(* Logix 5000 project; controller ABB_Drive_Test vendor 1 type 14 code 149 rev 33.12; software revision 33.01; part 6 of 6 *)
(* tags used below, declared in another part *)
   flagDesAcell : BOOL;   // Flag Auxiliar Boton de Parada
   indiceLocal : DINT;
   InicioDinagram : BOOL;   // Inicio de la Adquisión del Dinagrama
   numeroMuestras : DINT;   // Numero de Muestras del Stroke
   pausa : BOOL;
   rpmFeedback : INT;   // Valor absoluto de la referencia 0 no lo toma
   VCarga : REAL[1500];
   Vct : REAL[1500];
   VPosicion : REAL[1500];   // vector de potencia por comunicación
   VPotencia : REAL[1500];
   VPotenciaC : REAL[1500];   // Vector de potencia cableado
   VProximetro : BOOL[1504];
   ABB_GetAtt_Value : DINT;
   ABB_GetMsg : MESSAGE;
   ABB_Input : ABB_Read;
   ABB_Msg_SetValue : DINT;
   ABB_Output : ABB_Write;
   ABB_SetMsg : MESSAGE;
   counters : COUNTER[20];
   Proximetro : BOOL;
   SWC : SWC;
   Timmers : TIMER[10];
(* T000_MainProgram, continued *)

ROUTINE R001_ABB_Drive   (* ladder *)
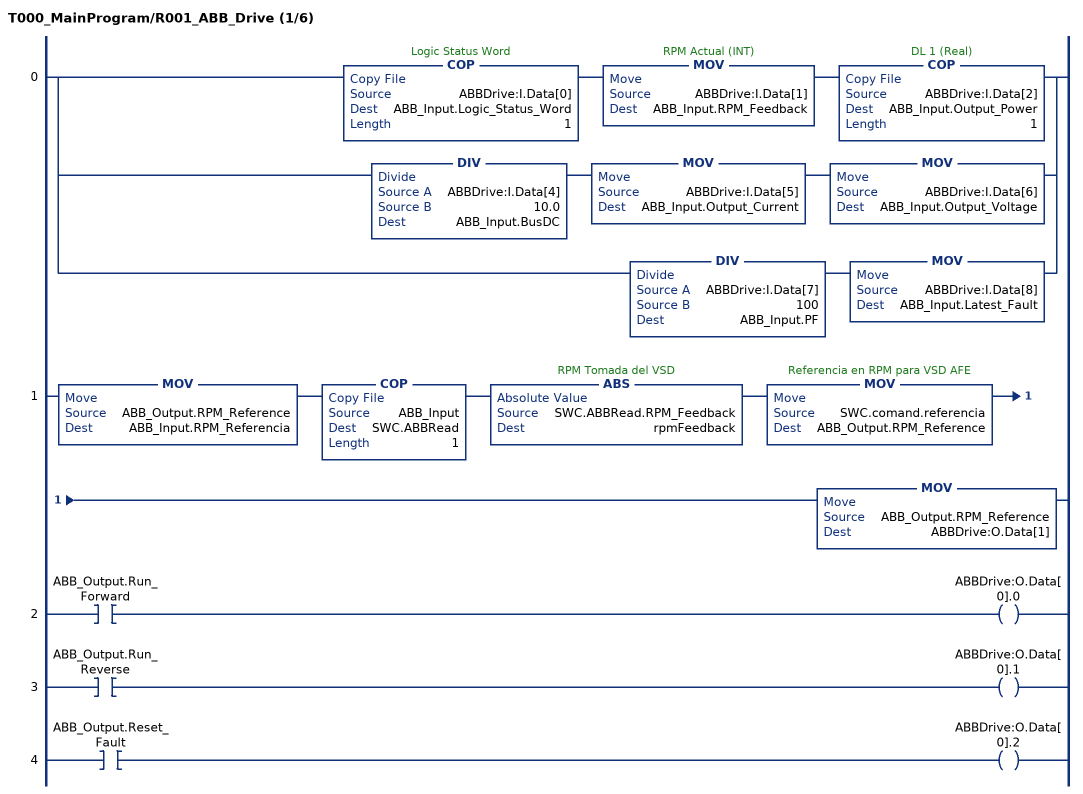
   0: [COP(ABBDrive:I.Data[0],ABB_Input.Logic_Status_Word,1) MOV(ABBDrive:I.Data[1],ABB_Input.RPM_Feedback) COP(ABBDrive:I.Data[2],ABB_Input.Output_Power,1) ,DIV(ABBDrive:I.Data[4],10.0,ABB_Input.BusDC) MOV(ABBDrive:I.Data[5],ABB_Input.Output_Current) MOV(ABBDrive:I.Data[6],ABB_Input.Output_Voltage) ,DIV(ABBDrive:I.Data[7],100,ABB_Input.PF) MOV(ABBDrive:I.Data[8],ABB_Input.Latest_Fault) ];
   1: MOV(ABB_Output.RPM_Reference,ABB_Input.RPM_Referencia)COP(ABB_Input,SWC.ABBRead,1)ABS(SWC.ABBRead.RPM_Feedback,rpmFeedback)MOV(SWC.comand.referencia,ABB_Output.RPM_Reference)MOV(ABB_Output.RPM_Reference,ABBDrive:O.Data[1]);
   2: XIC(ABB_Output.Run_Forward)OTE(ABBDrive:O.Data[0].0);
   3: XIC(ABB_Output.Run_Reverse)OTE(ABBDrive:O.Data[0].1);
   4: XIC(ABB_Output.Reset_Fault)OTE(ABBDrive:O.Data[0].2);
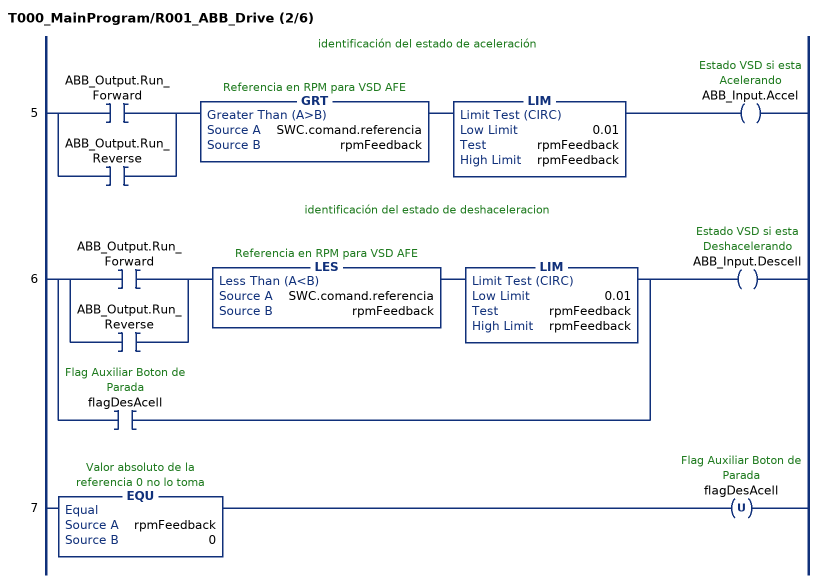
   // identificación del estado de aceleración
   5: [XIC(ABB_Output.Run_Forward) ,XIC(ABB_Output.Run_Reverse) ]GRT(SWC.comand.referencia,rpmFeedback)LIM(0.01,rpmFeedback,rpmFeedback)OTE(ABB_Input.Accel);
   // identificación del estado de deshaceleracion
   6: [[XIC(ABB_Output.Run_Forward) ,XIC(ABB_Output.Run_Reverse) ] LES(SWC.comand.referencia,rpmFeedback) LIM(0.01,rpmFeedback,rpmFeedback) ,XIC(flagDesAcell) ]OTE(ABB_Input.Descell);
   7: EQU(rpmFeedback,0)OTU(flagDesAcell);
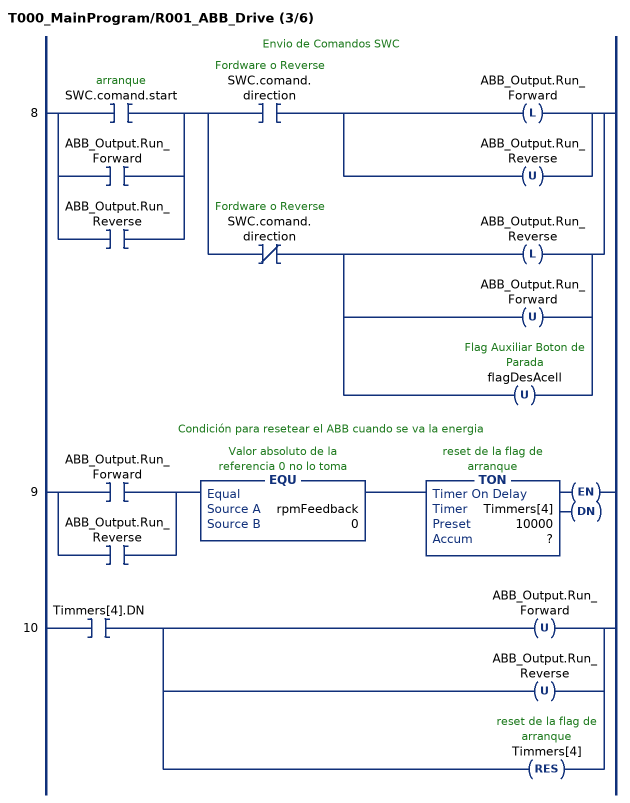
   // Envio de Comandos SWC
   8: [[XIC(SWC.comand.start) ,XIC(ABB_Output.Run_Forward) ] ,XIC(ABB_Output.Run_Reverse) ][XIC(SWC.comand.direction) [OTL(ABB_Output.Run_Forward) ,OTU(ABB_Output.Run_Reverse) ] ,XIO(SWC.comand.direction) [OTL(ABB_Output.Run_Reverse) ,[OTU(ABB_Output.Run_Forward) ,OTU(flagDesAcell) ] ] ];
   // Condición para resetear el ABB cuando se va la energia
   9: [XIC(ABB_Output.Run_Forward) ,XIC(ABB_Output.Run_Reverse) ]EQU(rpmFeedback,0)TON(Timmers[4],?,?);
   10: XIC(Timmers[4].DN)[OTU(ABB_Output.Run_Forward) ,[OTU(ABB_Output.Run_Reverse) ,RES(Timmers[4]) ] ];
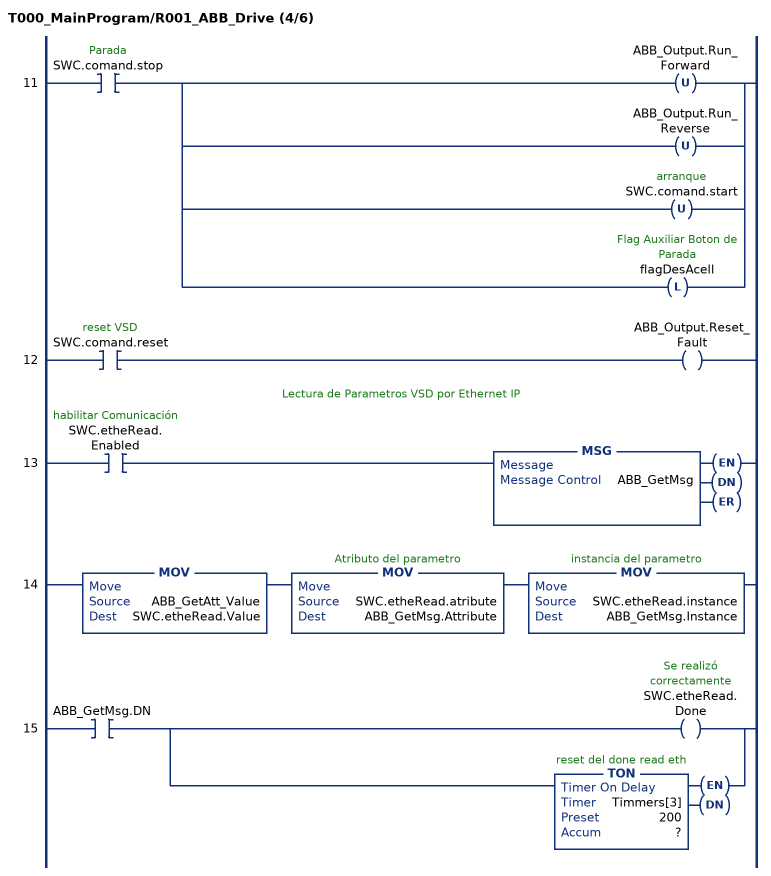
   11: XIC(SWC.comand.stop)[OTU(ABB_Output.Run_Forward) ,[OTU(ABB_Output.Run_Reverse) ,[OTU(SWC.comand.start) ,OTL(flagDesAcell) ] ] ];
   12: XIC(SWC.comand.reset)OTE(ABB_Output.Reset_Fault);
   // Lectura de Parametros VSD por Ethernet IP
   13: XIC(SWC.etheRead.Enabled)MSG(ABB_GetMsg);
   14: MOV(ABB_GetAtt_Value,SWC.etheRead.Value)MOV(SWC.etheRead.atribute,ABB_GetMsg.Attribute)MOV(SWC.etheRead.instance,ABB_GetMsg.Instance);
   15: XIC(ABB_GetMsg.DN)[OTE(SWC.etheRead.Done) ,TON(Timmers[3],?,?) ];
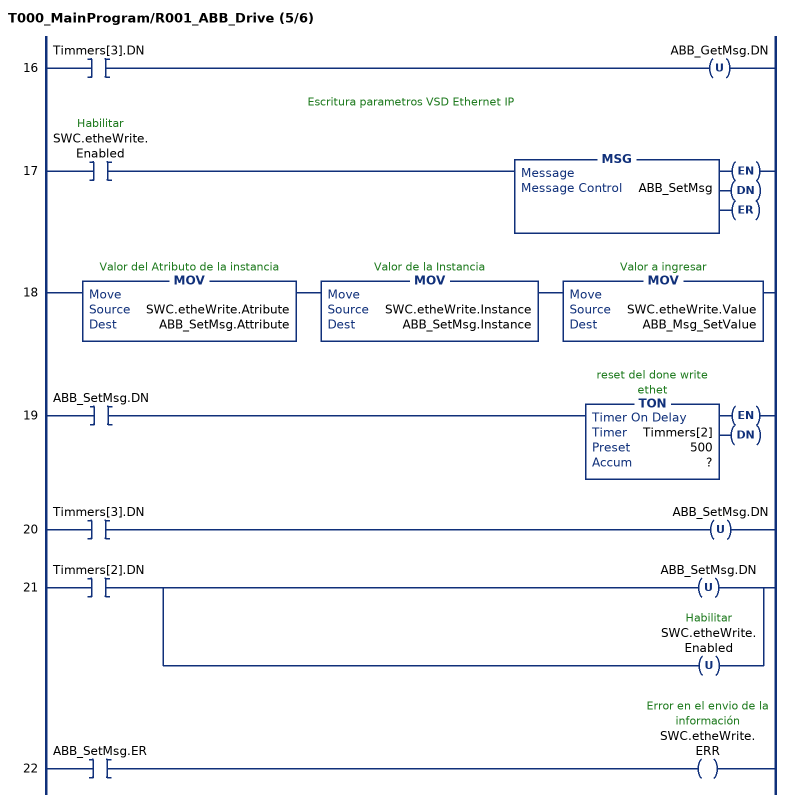
   16: XIC(Timmers[3].DN)OTU(ABB_GetMsg.DN);
   // Escritura parametros VSD Ethernet IP
   17: XIC(SWC.etheWrite.Enabled)MSG(ABB_SetMsg);
   18: MOV(SWC.etheWrite.Atribute,ABB_SetMsg.Attribute)MOV(SWC.etheWrite.Instance,ABB_SetMsg.Instance)MOV(SWC.etheWrite.Value,ABB_Msg_SetValue);
   19: XIC(ABB_SetMsg.DN)TON(Timmers[2],?,?);
   20: XIC(Timmers[3].DN)OTU(ABB_SetMsg.DN);
   21: XIC(Timmers[2].DN)[OTU(ABB_SetMsg.DN) ,OTU(SWC.etheWrite.Enabled) ];
   22: XIC(ABB_SetMsg.ER)OTE(SWC.etheWrite.ERR);
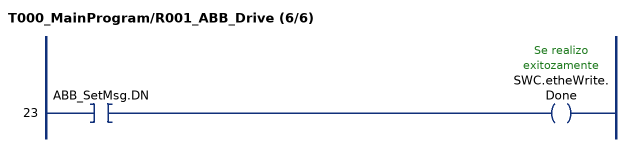
   23: XIC(ABB_SetMsg.DN)OTE(SWC.etheWrite.Done);
END_ROUTINE

ROUTINE R002_Dinagram   (* ladder *)
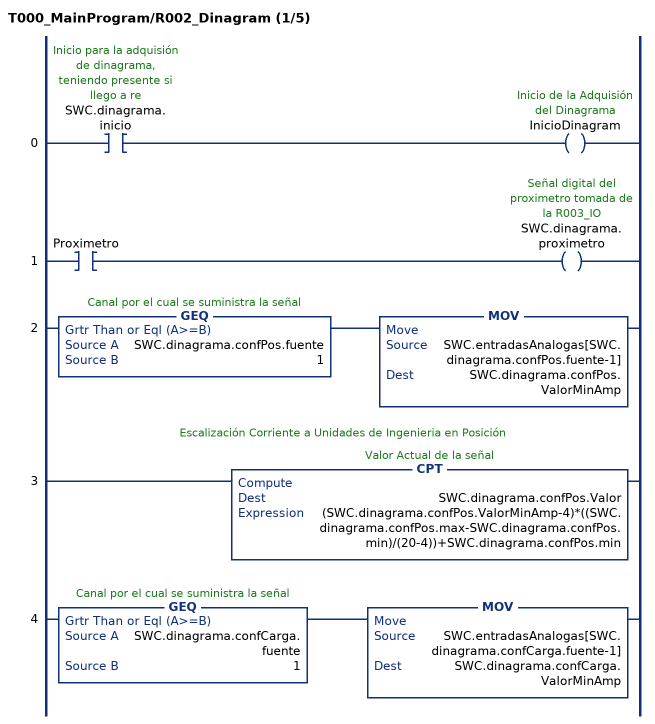
   0: XIC(SWC.dinagrama.inicio)OTE(InicioDinagram);
   1: XIC(Proximetro)OTE(SWC.dinagrama.proximetro);
   2: GEQ(SWC.dinagrama.confPos.fuente,1)MOV(SWC.entradasAnalogas[SWC.dinagrama.confPos.fuente-1],SWC.dinagrama.confPos.ValorMinAmp);
   // Escalización Corriente a Unidades de Ingenieria en Posición
   3: CPT(SWC.dinagrama.confPos.Valor,(SWC.dinagrama.confPos.ValorMinAmp-4)*((SWC.dinagrama.confPos.max-SWC.dinagrama.confPos.min)/(20-4))+SWC.dinagrama.confPos.min);
   4: GEQ(SWC.dinagrama.confCarga.fuente,1)MOV(SWC.entradasAnalogas[SWC.dinagrama.confCarga.fuente-1],SWC.dinagrama.confCarga.ValorMinAmp);
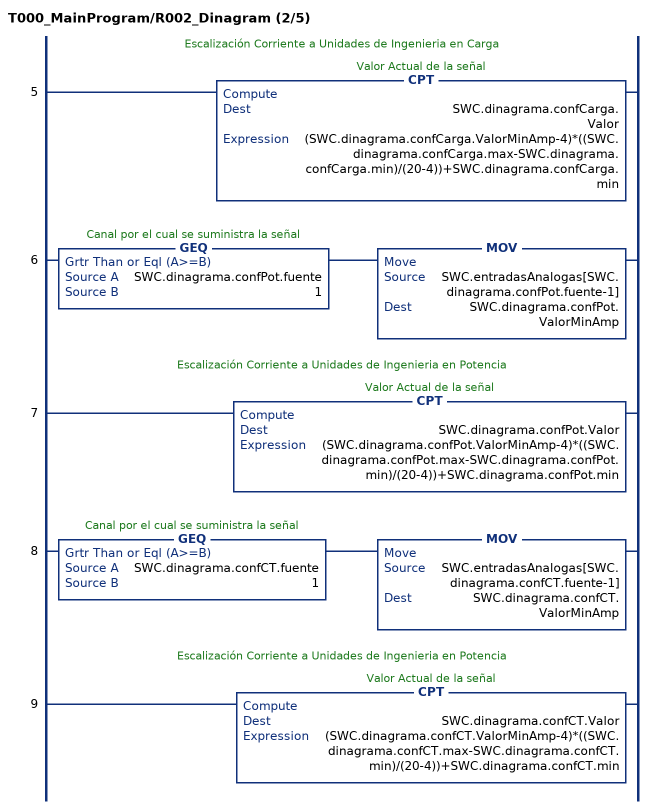
   // Escalización Corriente a Unidades de Ingenieria en Carga
   5: CPT(SWC.dinagrama.confCarga.Valor,(SWC.dinagrama.confCarga.ValorMinAmp-4)*((SWC.dinagrama.confCarga.max-SWC.dinagrama.confCarga.min)/(20-4))+SWC.dinagrama.confCarga.min);
   6: GEQ(SWC.dinagrama.confPot.fuente,1)MOV(SWC.entradasAnalogas[SWC.dinagrama.confPot.fuente-1],SWC.dinagrama.confPot.ValorMinAmp);
   // Escalización Corriente a Unidades de Ingenieria en Potencia
   7: CPT(SWC.dinagrama.confPot.Valor,(SWC.dinagrama.confPot.ValorMinAmp-4)*((SWC.dinagrama.confPot.max-SWC.dinagrama.confPot.min)/(20-4))+SWC.dinagrama.confPot.min);
   8: GEQ(SWC.dinagrama.confCT.fuente,1)MOV(SWC.entradasAnalogas[SWC.dinagrama.confCT.fuente-1],SWC.dinagrama.confCT.ValorMinAmp);
   // Escalización Corriente a Unidades de Ingenieria en Potencia
   9: CPT(SWC.dinagrama.confCT.Valor,(SWC.dinagrama.confCT.ValorMinAmp-4)*((SWC.dinagrama.confCT.max-SWC.dinagrama.confCT.min)/(20-4))+SWC.dinagrama.confCT.min);
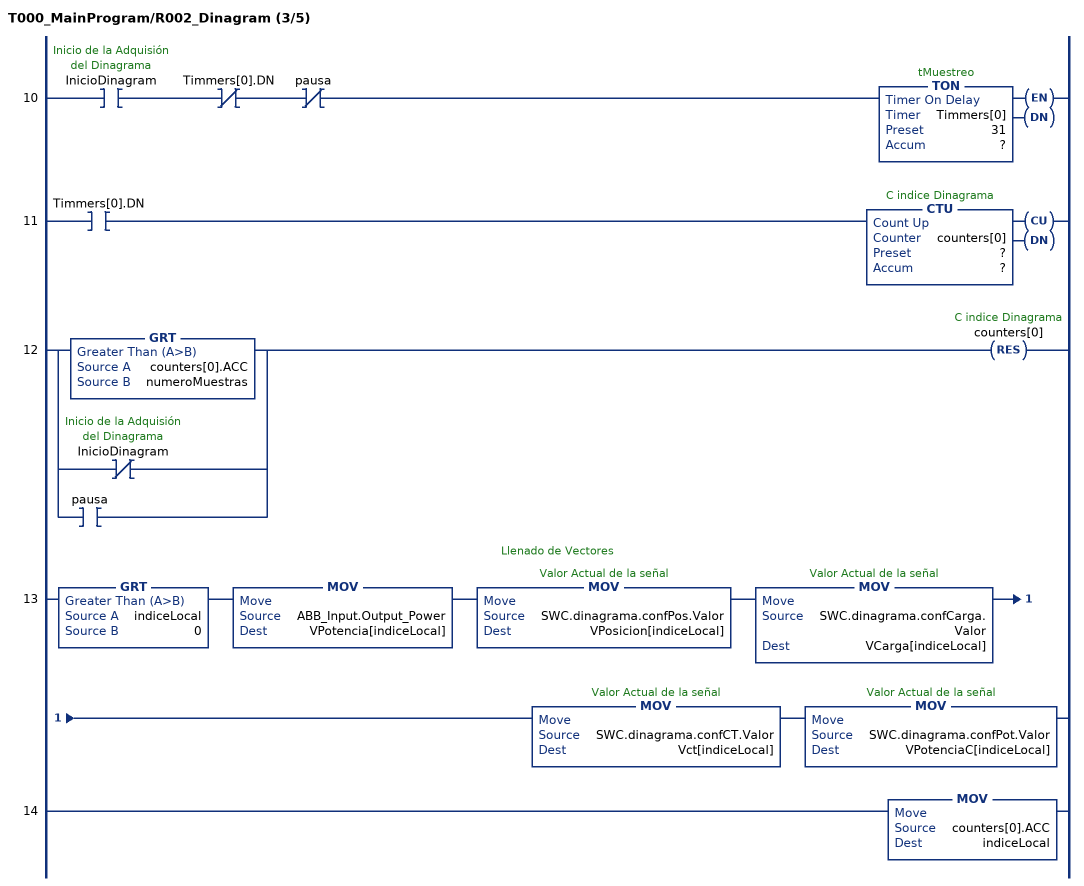
   10: XIC(InicioDinagram)XIO(Timmers[0].DN)XIO(pausa)TON(Timmers[0],?,?);
   11: XIC(Timmers[0].DN)CTU(counters[0],?,?);
   12: [[GRT(counters[0].ACC,numeroMuestras) ,XIO(InicioDinagram) ] ,XIC(pausa) ]RES(counters[0]);
   // Llenado de Vectores
   13: GRT(indiceLocal,0)MOV(ABB_Input.Output_Power,VPotencia[indiceLocal])MOV(SWC.dinagrama.confPos.Valor,VPosicion[indiceLocal])MOV(SWC.dinagrama.confCarga.Valor,VCarga[indiceLocal])MOV(SWC.dinagrama.confCT.Valor,Vct[indiceLocal])MOV(SWC.dinagrama.confPot.Valor,VPotenciaC[indiceLocal]);
   14: MOV(counters[0].ACC,indiceLocal);
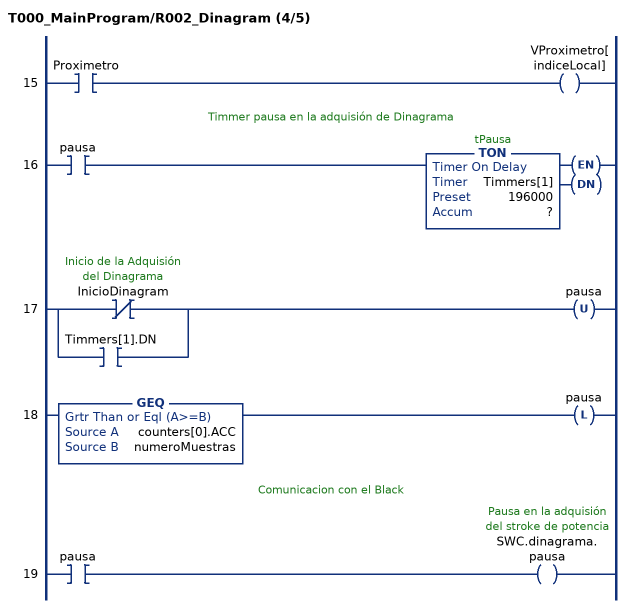
   15: XIC(Proximetro)OTE(VProximetro[indiceLocal]);
   // Timmer pausa en la adquisión de Dinagrama
   16: XIC(pausa)TON(Timmers[1],?,?);
   17: [XIO(InicioDinagram) ,XIC(Timmers[1].DN) ]OTU(pausa);
   18: GEQ(counters[0].ACC,numeroMuestras)OTL(pausa);
   // Comunicacion con el Black
   19: XIC(pausa)OTE(SWC.dinagrama.pausa);
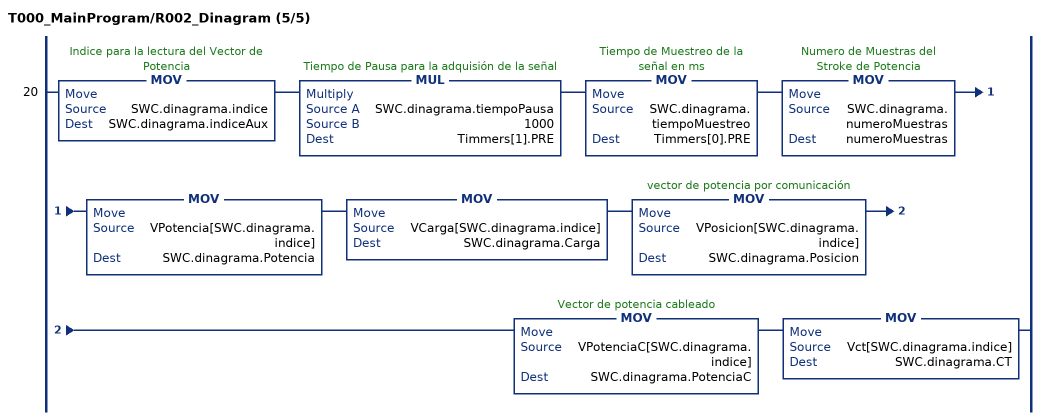
   20: MOV(SWC.dinagrama.indice,SWC.dinagrama.indiceAux)MUL(SWC.dinagrama.tiempoPausa,1000,Timmers[1].PRE)MOV(SWC.dinagrama.tiempoMuestreo,Timmers[0].PRE)MOV(SWC.dinagrama.numeroMuestras,numeroMuestras)MOV(VPotencia[SWC.dinagrama.indice],SWC.dinagrama.Potencia)MOV(VCarga[SWC.dinagrama.indice],SWC.dinagrama.Carga)MOV(VPosicion[SWC.dinagrama.indice],SWC.dinagrama.Posicion)MOV(VPotenciaC[SWC.dinagrama.indice],SWC.dinagrama.PotenciaC)MOV(Vct[SWC.dinagrama.indice],SWC.dinagrama.CT);
END_ROUTINE

ROUTINE R003_IO_Digital   (* ladder *)
// Entradas Digitales
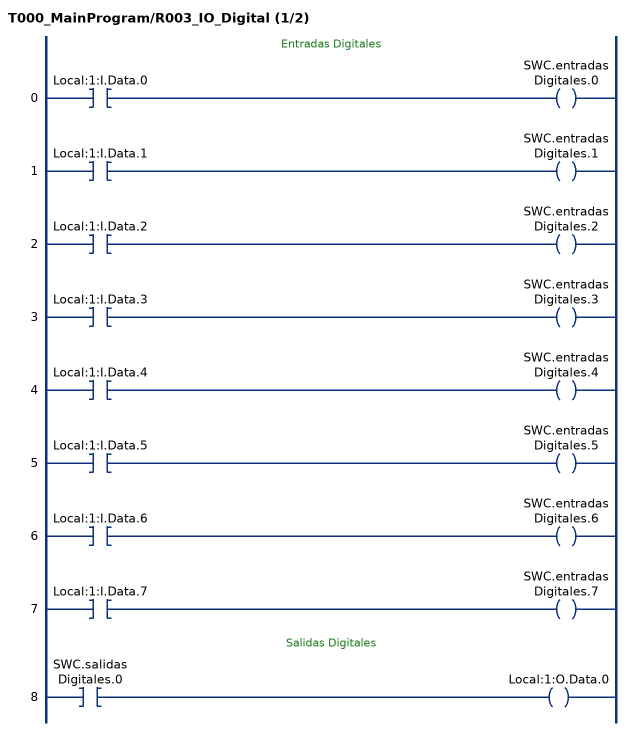
   // Entradas Digitales
   0: XIC(Local:1:I.Data.0)OTE(SWC.entradasDigitales.0);
   1: XIC(Local:1:I.Data.1)OTE(SWC.entradasDigitales.1);
   2: XIC(Local:1:I.Data.2)OTE(SWC.entradasDigitales.2);
   3: XIC(Local:1:I.Data.3)OTE(SWC.entradasDigitales.3);
   4: XIC(Local:1:I.Data.4)OTE(SWC.entradasDigitales.4);
   5: XIC(Local:1:I.Data.5)OTE(SWC.entradasDigitales.5);
   6: XIC(Local:1:I.Data.6)OTE(SWC.entradasDigitales.6);
   7: XIC(Local:1:I.Data.7)OTE(SWC.entradasDigitales.7);
   // Salidas Digitales
   8: XIC(SWC.salidasDigitales.0)OTE(Local:1:O.Data.0);
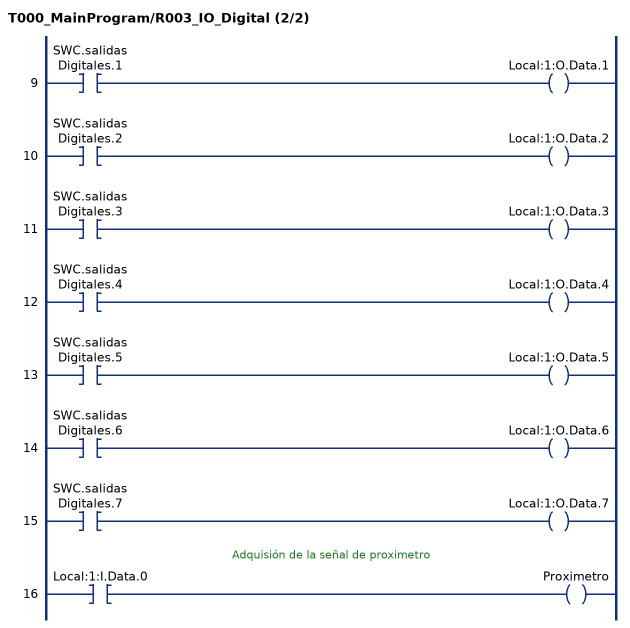
   9: XIC(SWC.salidasDigitales.1)OTE(Local:1:O.Data.1);
   10: XIC(SWC.salidasDigitales.2)OTE(Local:1:O.Data.2);
   11: XIC(SWC.salidasDigitales.3)OTE(Local:1:O.Data.3);
   12: XIC(SWC.salidasDigitales.4)OTE(Local:1:O.Data.4);
   13: XIC(SWC.salidasDigitales.5)OTE(Local:1:O.Data.5);
   14: XIC(SWC.salidasDigitales.6)OTE(Local:1:O.Data.6);
   15: XIC(SWC.salidasDigitales.7)OTE(Local:1:O.Data.7);
   // Adquisión de la señal de proximetro
   16: XIC(Local:1:I.Data.0)OTE(Proximetro);
END_ROUTINE

ROUTINE R004_IO_Anologica   (* function block diagram *)
// Rutina Para Entradas  Analogas
   SHEET 1
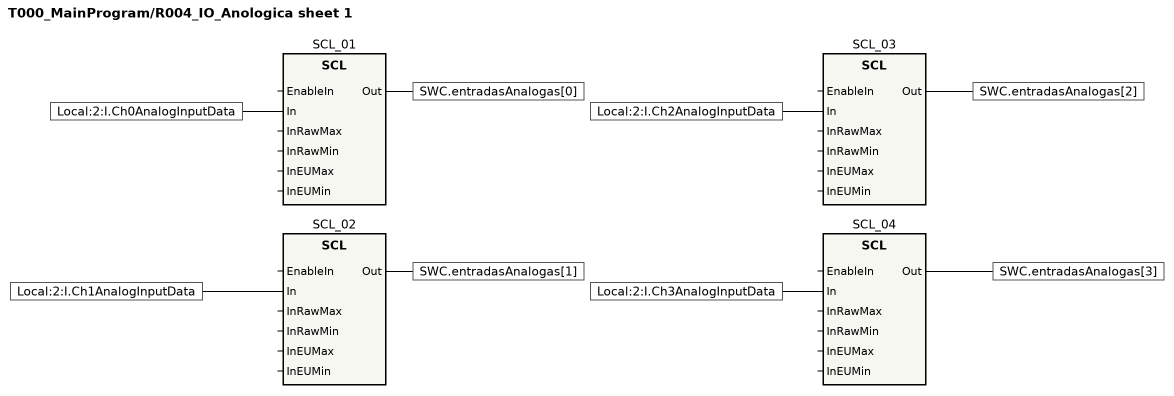
   SCL_01 : SCL(In := Local:2:I.Ch0AnalogInputData);   // unwired pins: EnableIn InRawMax InRawMin InEUMax InEUMin
   SCL_02 : SCL(In := Local:2:I.Ch1AnalogInputData);   // unwired pins: EnableIn InRawMax InRawMin InEUMax InEUMin
   SWC.entradasAnalogas[0] := SCL_01.Out;
   SWC.entradasAnalogas[1] := SCL_02.Out;
   SCL_03 : SCL(In := Local:2:I.Ch2AnalogInputData);   // unwired pins: EnableIn InRawMax InRawMin InEUMax InEUMin
   SCL_04 : SCL(In := Local:2:I.Ch3AnalogInputData);   // unwired pins: EnableIn InRawMax InRawMin InEUMax InEUMin
   SWC.entradasAnalogas[2] := SCL_03.Out;
   SWC.entradasAnalogas[3] := SCL_04.Out;
END_ROUTINE

ROUTINE R00_MainRoutine   (* ladder *)
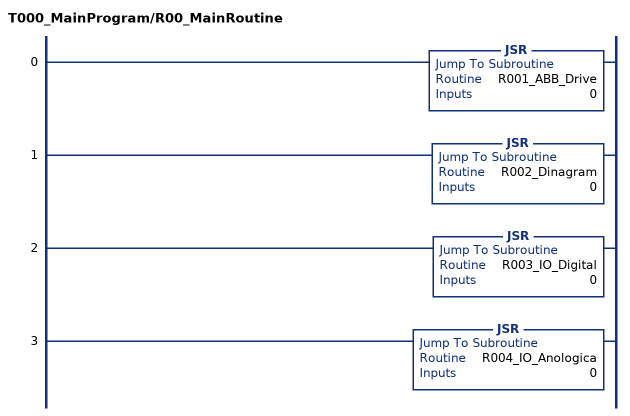
   0: JSR(R001_ABB_Drive,0);
   1: JSR(R002_Dinagram,0);
   2: JSR(R003_IO_Digital,0);
   3: JSR(R004_IO_Anologica,0);
END_ROUTINE
END_PROGRAM
